{attribute 'pack_mode' := '1'}
TYPE ST_Siemens_RcvDp_Status :
STRUCT
	nSendData				: WORD;
	nSendSequenceNumber		: WORD;	
	nSendCrc				: WORD;
END_STRUCT
END_TYPE

(* stored: Version 1.1.0.1, ProductVersion 3.1.4024.12
   DUT ST_Siemens_RcvDp_Status: Id {e5844c80-7a99-0882-00ef-ddd2ff196a0e} *)
